SUBAPPLICATION Uebung_053 (* DigitalInput_I1-_I4 auf DigitalOutput_Q1-_Q4 *)
  (* Standard: 61499-2; Description: Copyright (c) 2023 Meisterschulen am Ostbahnhof This program and the accompanying materials are made available under the terms of the Eclipse Public License 2.0 which is available at https://www.eclipse.org/legal/epl-2.0/ SPDX-License-Identifier: EPL-2.0 *)
  (* Version 1.0, 2023-10-23, Franz Höpfinger, Meisterschulen am Ostbahnhof *)
  PACKAGE Uebungen;
  IMPORT logiBUS::io::DI::logiBUS_DI::Input_I1;
  IMPORT logiBUS::io::DI::logiBUS_DI::Input_I2;
  IMPORT logiBUS::io::DI::logiBUS_DI::Input_I3;
  IMPORT logiBUS::io::DI::logiBUS_DI::Input_I4;
  IMPORT logiBUS::io::DQ::logiBUS_DO::Output_Q1;
  IMPORT logiBUS::io::DQ::logiBUS_DO::Output_Q2;
  IMPORT logiBUS::io::DQ::logiBUS_DO::Output_Q3;
  IMPORT logiBUS::io::DQ::logiBUS_DO::Output_Q4;
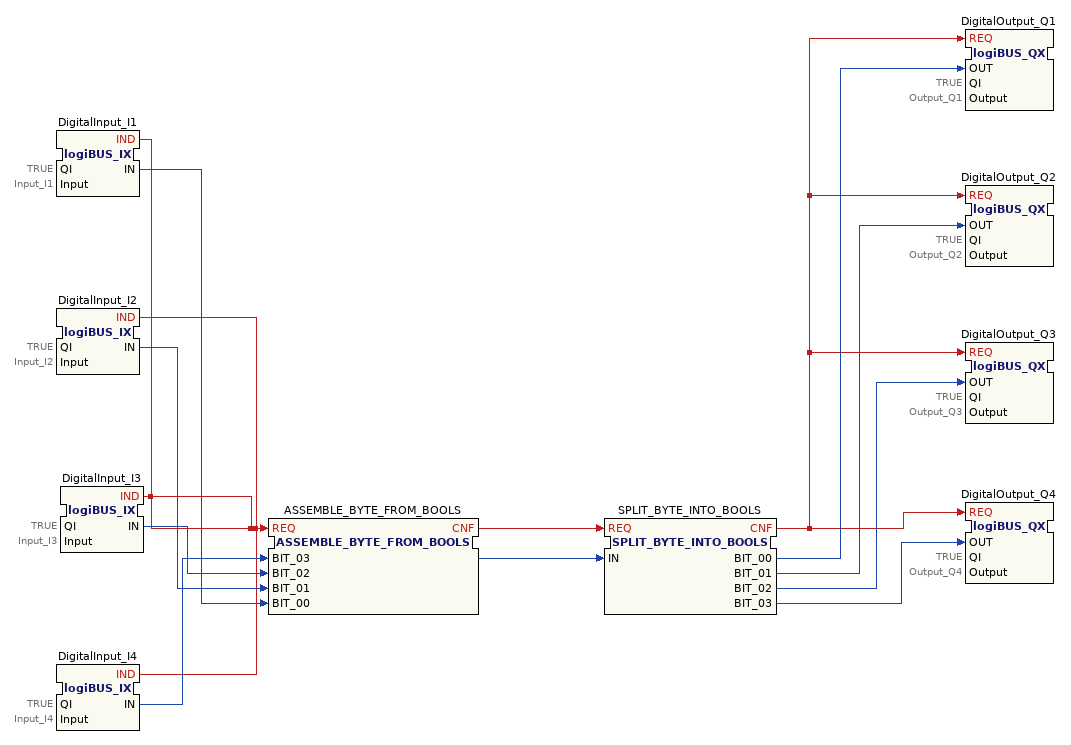
  FBS
    DigitalOutput_Q1 : logiBUS::io::DQ::logiBUS_QX(QI := TRUE, Output := Output_Q1);
    DigitalInput_I1 : logiBUS::io::DI::logiBUS_IX(QI := TRUE, Input := Input_I1);
    DigitalOutput_Q2 : logiBUS::io::DQ::logiBUS_QX(QI := TRUE, Output := Output_Q2);
    DigitalInput_I2 : logiBUS::io::DI::logiBUS_IX(QI := TRUE, Input := Input_I2);
    DigitalOutput_Q3 : logiBUS::io::DQ::logiBUS_QX(QI := TRUE, Output := Output_Q3);
    DigitalInput_I3 : logiBUS::io::DI::logiBUS_IX(QI := TRUE, Input := Input_I3);
    DigitalOutput_Q4 : logiBUS::io::DQ::logiBUS_QX(QI := TRUE, Output := Output_Q4);
    DigitalInput_I4 : logiBUS::io::DI::logiBUS_IX(QI := TRUE, Input := Input_I4);
    ASSEMBLE_BYTE_FROM_BOOLS : eclipse4diac::utils::assembling::ASSEMBLE_BYTE_FROM_BOOLS;
    SPLIT_BYTE_INTO_BOOLS : eclipse4diac::utils::splitting::SPLIT_BYTE_INTO_BOOLS;
  END_FBS
  EVENT_CONNECTIONS
    ASSEMBLE_BYTE_FROM_BOOLS.CNF TO SPLIT_BYTE_INTO_BOOLS.REQ;
    DigitalInput_I1.IND TO ASSEMBLE_BYTE_FROM_BOOLS.REQ;
    DigitalInput_I2.IND TO ASSEMBLE_BYTE_FROM_BOOLS.REQ;
    DigitalInput_I3.IND TO ASSEMBLE_BYTE_FROM_BOOLS.REQ;
    DigitalInput_I4.IND TO ASSEMBLE_BYTE_FROM_BOOLS.REQ;
    SPLIT_BYTE_INTO_BOOLS.CNF TO DigitalOutput_Q1.REQ;
    SPLIT_BYTE_INTO_BOOLS.CNF TO DigitalOutput_Q2.REQ;
    SPLIT_BYTE_INTO_BOOLS.CNF TO DigitalOutput_Q3.REQ;
    SPLIT_BYTE_INTO_BOOLS.CNF TO DigitalOutput_Q4.REQ;
  END_CONNECTIONS
  DATA_CONNECTIONS
    ASSEMBLE_BYTE_FROM_BOOLS. TO SPLIT_BYTE_INTO_BOOLS.IN;
    SPLIT_BYTE_INTO_BOOLS.BIT_00 TO DigitalOutput_Q1.OUT;
    SPLIT_BYTE_INTO_BOOLS.BIT_01 TO DigitalOutput_Q2.OUT;
    SPLIT_BYTE_INTO_BOOLS.BIT_02 TO DigitalOutput_Q3.OUT;
    SPLIT_BYTE_INTO_BOOLS.BIT_03 TO DigitalOutput_Q4.OUT;
    DigitalInput_I4.IN TO ASSEMBLE_BYTE_FROM_BOOLS.BIT_03;
    DigitalInput_I3.IN TO ASSEMBLE_BYTE_FROM_BOOLS.BIT_02;
    DigitalInput_I2.IN TO ASSEMBLE_BYTE_FROM_BOOLS.BIT_01;
    DigitalInput_I1.IN TO ASSEMBLE_BYTE_FROM_BOOLS.BIT_00;
  END_CONNECTIONS
END_SUBAPPLICATION
